// TIA Portal V20 export
FUNCTION_BLOCK "LER_EQP_Interface_OtherStack"   // FB141, LAD
// stored: Access Published, MemoryReserve 100, SetENOAutomatically false
   VAR_INPUT
      enable : Bool;
      executeCmd : Bool;
      clock : Bool;
      heartBeat : Byte;
      unitStatus : "LAF_typeUnitStatus";
      unitAlarms : "LAF_typeAlarms";
   END_VAR
   VAR_OUTPUT
      error : Bool;
      status : Word;
   END_VAR
   VAR_IN_OUT
      StackCommunication : "LER_typeCommunicationStack";
      MotionStatus : "LER_typeCommonDataStackMotion";
      configuration : "LER_typeCommunicationConfiguration";
      moduleInterface : "LER_typeCommunicationInterface";
      controlNode : "LER_typeCommunicationControlNode";
   END_VAR
   VAR
      instEQP_Interface_Communication { S7_SetPoint := 'True'} : "LER_EQP_Communication";
      statInsHeartBeat : Byte;
      statStackState : Struct
         Stop : Bool;
         Abort : Bool;
         Hold : Bool;
         Complete : Bool;
         Idle : Bool;
         TotalStop : Bool;
      END_STRUCT;
      statTonTimer : Array[0..9] of TON_TIME;
      statTofTimer : Array[0..9] of TOF_TIME;
   END_VAR
   VAR CONSTANT
      STATUS_NO_ERROR_OCCURRED : Word := 16#0;
      ERR_HEARTBEAT_ERROR : Word := 16#8000;
   END_VAR
BEGIN

REGION Network 1: EQP Interface Stack State
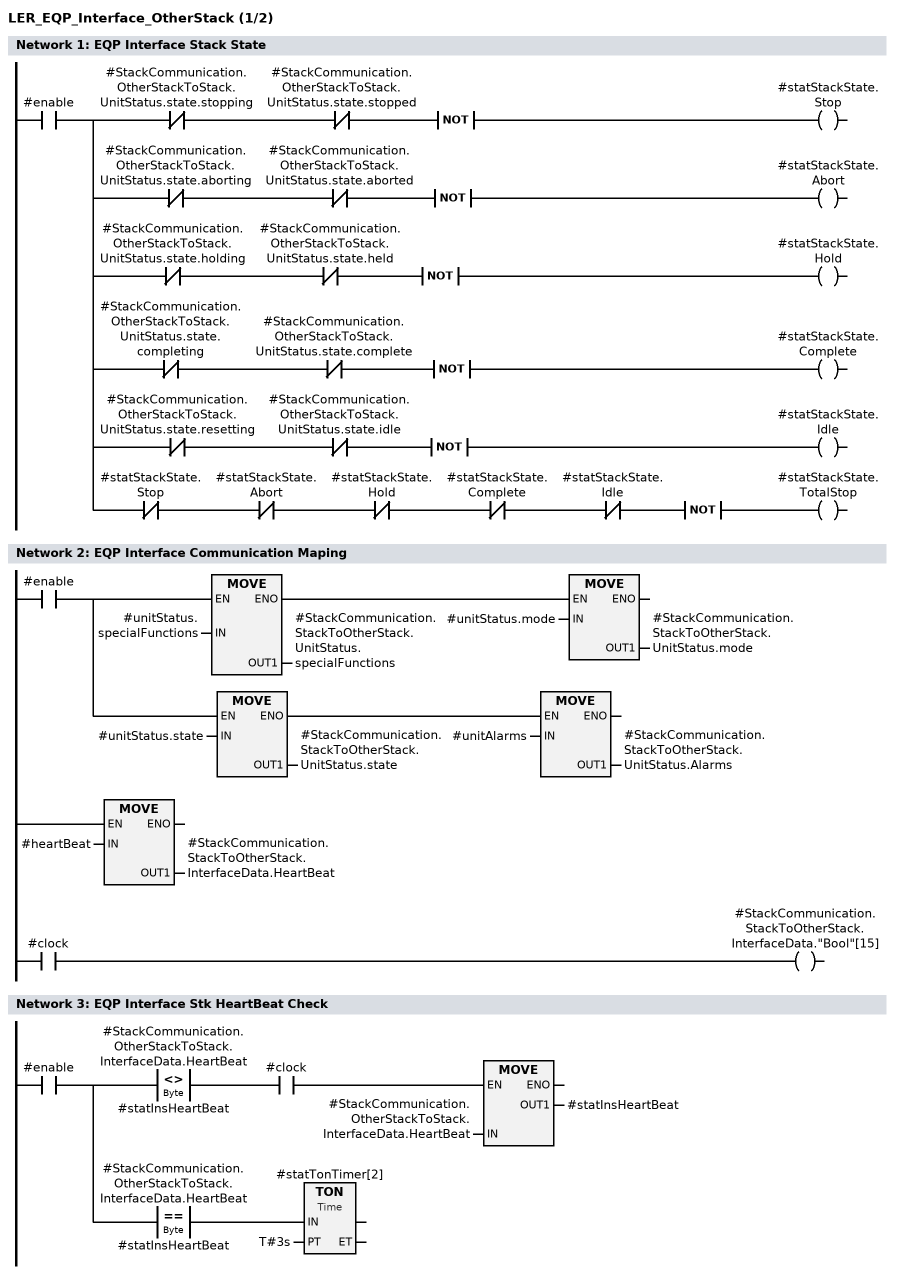
   RUNG wire#powerrail
      Contact( #enable )
      wire#w1
      I_Contact( #StackCommunication.OtherStackToStack.UnitStatus.state.stopping )
      I_Contact( #StackCommunication.OtherStackToStack.UnitStatus.state.stopped )
      Not()
      Coil( #statStackState.Stop )
   END_RUNG
   RUNG wire#w1
      I_Contact( #StackCommunication.OtherStackToStack.UnitStatus.state.aborting )
      I_Contact( #StackCommunication.OtherStackToStack.UnitStatus.state.aborted )
      Not()
      Coil( #statStackState.Abort )
   END_RUNG
   RUNG wire#w1
      I_Contact( #StackCommunication.OtherStackToStack.UnitStatus.state.holding )
      I_Contact( #StackCommunication.OtherStackToStack.UnitStatus.state.held )
      Not()
      Coil( #statStackState.Hold )
   END_RUNG
   RUNG wire#w1
      I_Contact( #StackCommunication.OtherStackToStack.UnitStatus.state.completing )
      I_Contact( #StackCommunication.OtherStackToStack.UnitStatus.state.complete )
      Not()
      Coil( #statStackState.Complete )
   END_RUNG
   RUNG wire#w1
      I_Contact( #StackCommunication.OtherStackToStack.UnitStatus.state.resetting )
      I_Contact( #StackCommunication.OtherStackToStack.UnitStatus.state.idle )
      Not()
      Coil( #statStackState.Idle )
   END_RUNG
   RUNG wire#w1
      I_Contact( #statStackState.Stop )
      I_Contact( #statStackState.Abort )
      I_Contact( #statStackState.Hold )
      I_Contact( #statStackState.Complete )
      I_Contact( #statStackState.Idle )
      Not()
      Coil( #statStackState.TotalStop )
   END_RUNG
   // the same network as SCL:
   #statStackState.Stop := NOT (#enable AND NOT #StackCommunication.OtherStackToStack.UnitStatus.state.stopping AND NOT #StackCommunication.OtherStackToStack.UnitStatus.state.stopped);
   #statStackState.Abort := NOT (#enable AND NOT #StackCommunication.OtherStackToStack.UnitStatus.state.aborting AND NOT #StackCommunication.OtherStackToStack.UnitStatus.state.aborted);
   #statStackState.Hold := NOT (#enable AND NOT #StackCommunication.OtherStackToStack.UnitStatus.state.holding AND NOT #StackCommunication.OtherStackToStack.UnitStatus.state.held);
   #statStackState.Complete := NOT (#enable AND NOT #StackCommunication.OtherStackToStack.UnitStatus.state.completing AND NOT #StackCommunication.OtherStackToStack.UnitStatus.state.complete);
   #statStackState.Idle := NOT (#enable AND NOT #StackCommunication.OtherStackToStack.UnitStatus.state.resetting AND NOT #StackCommunication.OtherStackToStack.UnitStatus.state.idle);
   #statStackState.TotalStop := NOT (#enable AND NOT #statStackState.Stop AND NOT #statStackState.Abort AND NOT #statStackState.Hold AND NOT #statStackState.Complete AND NOT #statStackState.Idle);
END_REGION

REGION Network 2: EQP Interface Communication Maping
   RUNG wire#powerrail
      Contact( #enable )
      wire#w1
      Move(in := #unitStatus.specialFunctions, out1 => #StackCommunication.StackToOtherStack.UnitStatus.specialFunctions)
      Move(in := #unitStatus.mode, out1 => #StackCommunication.StackToOtherStack.UnitStatus.mode)
   END_RUNG
   RUNG wire#w1
      Move(in := #unitStatus.state, out1 => #StackCommunication.StackToOtherStack.UnitStatus.state)
      Move(in := #unitAlarms, out1 => #StackCommunication.StackToOtherStack.UnitStatus.Alarms)
   END_RUNG
   RUNG wire#powerrail
      Move(in := #heartBeat, out1 => #StackCommunication.StackToOtherStack.InterfaceData.HeartBeat)
   END_RUNG
   RUNG wire#powerrail
      Contact( #clock )
      Coil( #StackCommunication.StackToOtherStack.InterfaceData."Bool"[15] )
   END_RUNG
   // the same network as SCL:
   IF #enable THEN
       #StackCommunication.StackToOtherStack.UnitStatus.specialFunctions := #unitStatus.specialFunctions;
       #StackCommunication.StackToOtherStack.UnitStatus.mode := #unitStatus.mode;
       #StackCommunication.StackToOtherStack.UnitStatus.state := #unitStatus.state;
       #StackCommunication.StackToOtherStack.UnitStatus.Alarms := #unitAlarms;
   END_IF;
   #StackCommunication.StackToOtherStack.InterfaceData.HeartBeat := #heartBeat;
   #StackCommunication.StackToOtherStack.InterfaceData."Bool"[15] := #clock;
END_REGION

REGION Network 3: EQP Interface Stk HeartBeat Check
   RUNG wire#powerrail
      Contact( #enable )
      wire#w1
      { S7_Templates := "SrcType := Byte" } NE_Contact(in1 := #StackCommunication.OtherStackToStack.InterfaceData.HeartBeat, in2 := #statInsHeartBeat)
      Contact( #clock )
      Move(in := #StackCommunication.OtherStackToStack.InterfaceData.HeartBeat, out1 => #statInsHeartBeat)
   END_RUNG
   RUNG wire#w1
      { S7_Templates := "SrcType := Byte" } EQ_Contact(in1 := #StackCommunication.OtherStackToStack.InterfaceData.HeartBeat, in2 := #statInsHeartBeat)
      { S7_Templates := "time_type := Time" } #statTonTimer[2].TON(pt := T#3s, et =>)
   END_RUNG
   // the same network as SCL:
   IF #enable AND (#StackCommunication.OtherStackToStack.InterfaceData.HeartBeat <> #statInsHeartBeat) AND #clock THEN
       #statInsHeartBeat := #StackCommunication.OtherStackToStack.InterfaceData.HeartBeat;
   END_IF;
   #statTonTimer[2].TON(IN := #enable AND (#StackCommunication.OtherStackToStack.InterfaceData.HeartBeat = #statInsHeartBeat),
                        PT := T#3s);
END_REGION

REGION Network 4: EQP Interface Communication Stack <-> OtherStack
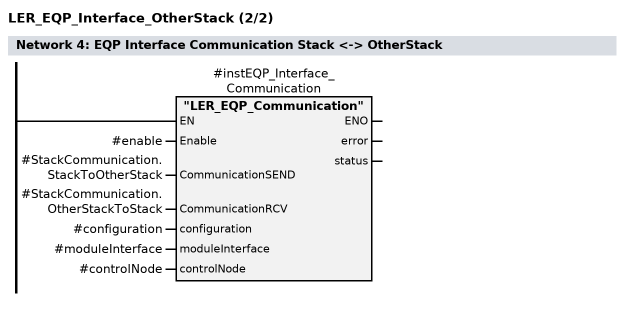
   RUNG wire#powerrail
      #instEQP_Interface_Communication(Enable := #enable, CommunicationSEND := #StackCommunication.StackToOtherStack, CommunicationRCV := #StackCommunication.OtherStackToStack, configuration := #configuration, moduleInterface := #moduleInterface, controlNode := #controlNode, error =>, status =>)
   END_RUNG
   // the same network as SCL:
   #instEQP_Interface_Communication(Enable := #enable,   // "LER_EQP_Communication"
                           CommunicationSEND := #StackCommunication.StackToOtherStack,
                           CommunicationRCV := #StackCommunication.OtherStackToStack,
                           configuration := #configuration,
                           moduleInterface := #moduleInterface,
                           controlNode := #controlNode);
END_REGION

REGION Network 5 (SCL): Error Check
   REGION Error Code Search

       IF #enable AND NOT #configuration.disableAlarms THEN
           IF #statTonTimer[2].Q THEN
               #status := #ERR_HEARTBEAT_ERROR;

           ELSIF #instEQP_Interface_Communication.error THEN
               #status := #instEQP_Interface_Communication.status;

           ELSE
               #status := #STATUS_NO_ERROR_OCCURRED;

           END_IF;
       ELSE
           #status := #STATUS_NO_ERROR_OCCURRED;

       END_IF;


       // Error Bit
       #error := #status <> 0;

   END_REGION
END_REGION

REGION Network 6 (SCL): ##### Outputs mapping #####
   #moduleInterface.monitoring.error := #error;
   #moduleInterface.monitoring.status := #status;

   #controlNode.monitoring := #moduleInterface.monitoring;
END_REGION
END_FUNCTION_BLOCK
